INTERFACE I_PackML_StoppedCommands

METHOD PUBLIC Abort
VAR_INPUT
END_VAR
END_METHOD

METHOD PUBLIC Reset
VAR_INPUT
END_VAR
END_METHOD

END_INTERFACE

(* stored: Version 1.1.0.1, ProductVersion 3.1.4024.12
   Itf I_PackML_StoppedCommands: Id {1719d416-8cac-0ada-1b61-0b25b7a48bba}
   Method Abort: Id {35195647-924b-054e-35e5-b1c69cbaa78e}
   Method Reset: Id {feb743ed-94f8-07ef-3bbd-fcb7c4d31c83} *)
